(* Logix 5000 project; controller SX_V040001_C001 vendor 1 type 14 code 77 rev 16.22; software revision 16.04; part 32 of 35 *)
(* tags used below, declared in another part *)
   ALL_KINDS : INT[90];
   PARAMETER : INT[501];
   pointer_recipe_test : DINT;
(* MainProgram, continued *)

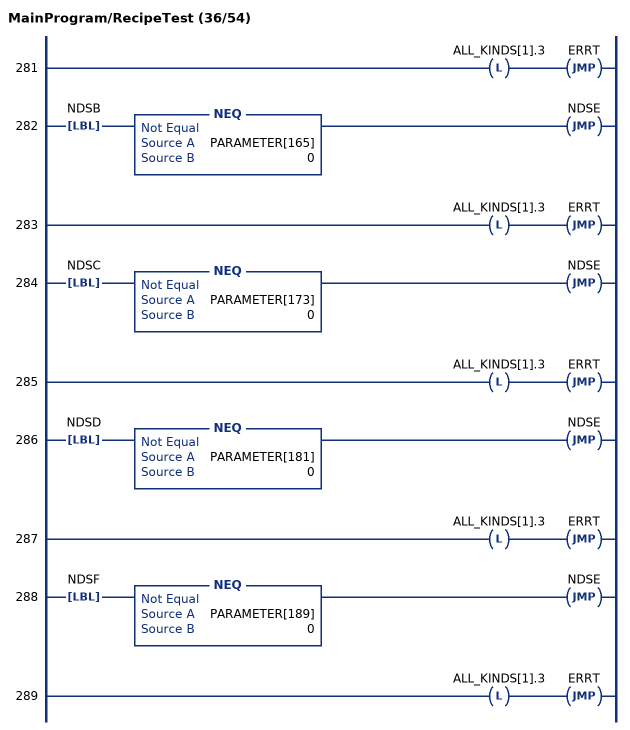
   [picture p701: MainProgram/RecipeTest rungs 281-289]
   281: OTL(ALL_KINDS[1].3)JMP(ERRT);
   282: LBL(NDSB)NEQ(PARAMETER[165],0)JMP(NDSE);
   283: OTL(ALL_KINDS[1].3)JMP(ERRT);
   284: LBL(NDSC)NEQ(PARAMETER[173],0)JMP(NDSE);
   285: OTL(ALL_KINDS[1].3)JMP(ERRT);
   286: LBL(NDSD)NEQ(PARAMETER[181],0)JMP(NDSE);
   287: OTL(ALL_KINDS[1].3)JMP(ERRT);
   288: LBL(NDSF)NEQ(PARAMETER[189],0)JMP(NDSE);
   289: OTL(ALL_KINDS[1].3)JMP(ERRT);
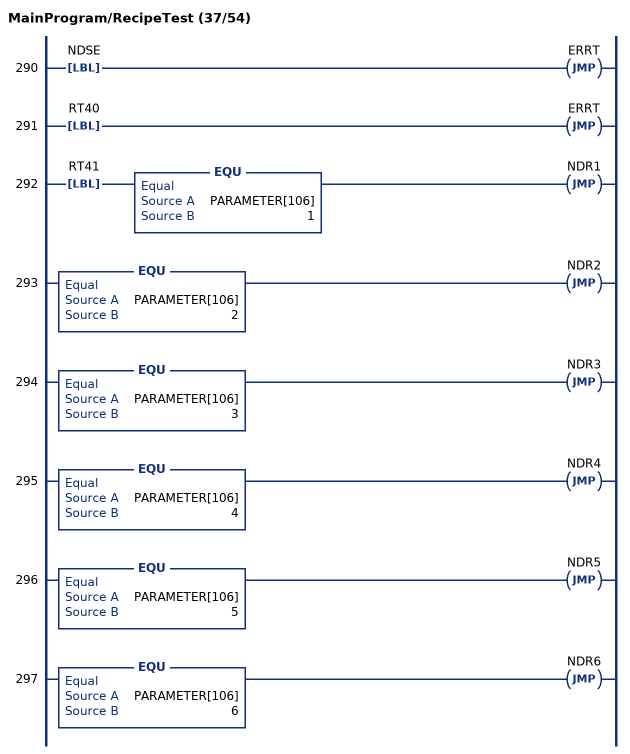
   290: LBL(NDSE)JMP(ERRT);
   291: LBL(RT40)JMP(ERRT);
   292: LBL(RT41)EQU(PARAMETER[106],1)JMP(NDR1);
   293: EQU(PARAMETER[106],2)JMP(NDR2);
   294: EQU(PARAMETER[106],3)JMP(NDR3);
   295: EQU(PARAMETER[106],4)JMP(NDR4);
   296: EQU(PARAMETER[106],5)JMP(NDR5);
   297: EQU(PARAMETER[106],6)JMP(NDR6);
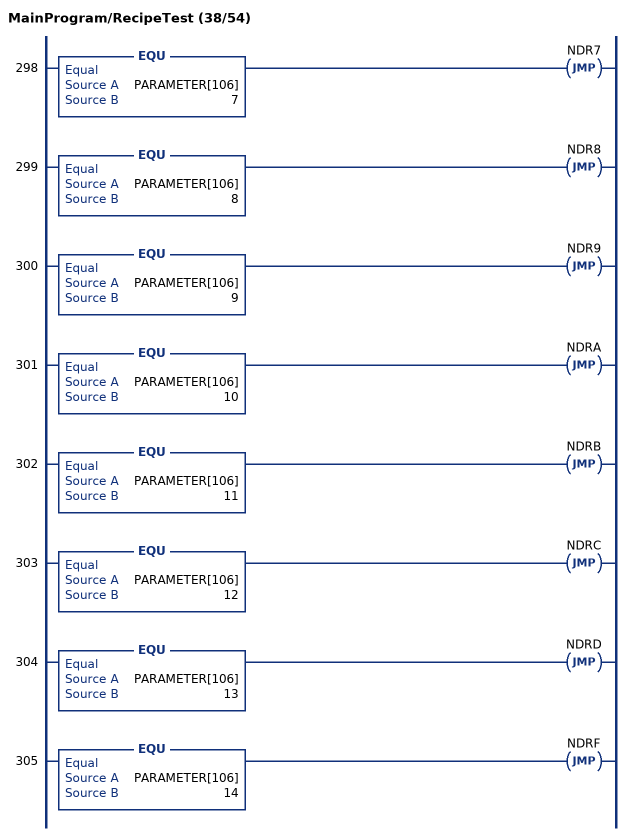
   298: EQU(PARAMETER[106],7)JMP(NDR7);
   299: EQU(PARAMETER[106],8)JMP(NDR8);
   300: EQU(PARAMETER[106],9)JMP(NDR9);
   301: EQU(PARAMETER[106],10)JMP(NDRA);
   302: EQU(PARAMETER[106],11)JMP(NDRB);
   303: EQU(PARAMETER[106],12)JMP(NDRC);
   304: EQU(PARAMETER[106],13)JMP(NDRD);
   305: EQU(PARAMETER[106],14)JMP(NDRF);
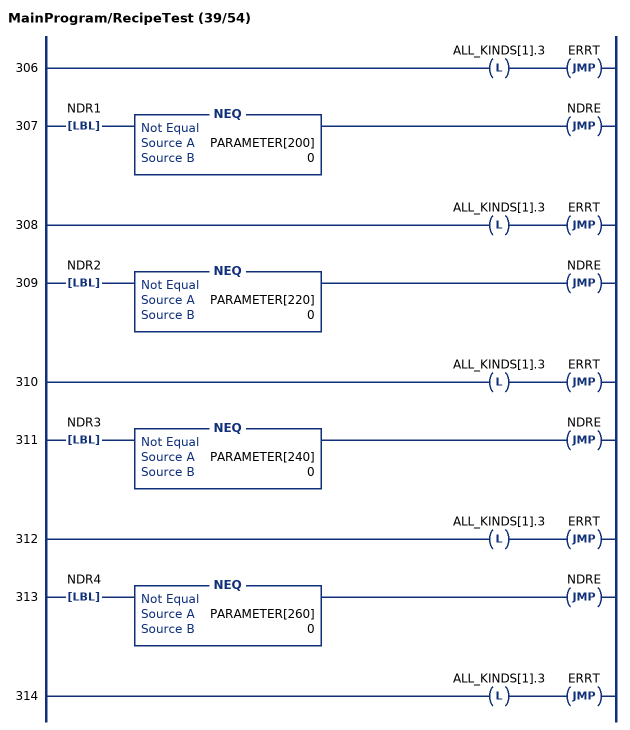
   306: OTL(ALL_KINDS[1].3)JMP(ERRT);
   307: LBL(NDR1)NEQ(PARAMETER[200],0)JMP(NDRE);
   308: OTL(ALL_KINDS[1].3)JMP(ERRT);
   309: LBL(NDR2)NEQ(PARAMETER[220],0)JMP(NDRE);
   310: OTL(ALL_KINDS[1].3)JMP(ERRT);
   311: LBL(NDR3)NEQ(PARAMETER[240],0)JMP(NDRE);
   312: OTL(ALL_KINDS[1].3)JMP(ERRT);
   313: LBL(NDR4)NEQ(PARAMETER[260],0)JMP(NDRE);
   314: OTL(ALL_KINDS[1].3)JMP(ERRT);
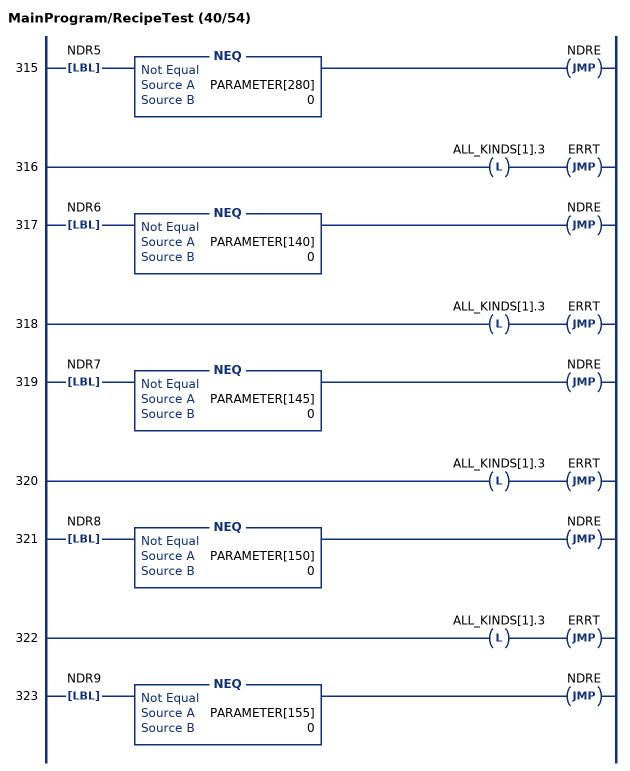
   315: LBL(NDR5)NEQ(PARAMETER[280],0)JMP(NDRE);
   316: OTL(ALL_KINDS[1].3)JMP(ERRT);
   317: LBL(NDR6)NEQ(PARAMETER[140],0)JMP(NDRE);
   318: OTL(ALL_KINDS[1].3)JMP(ERRT);
   319: LBL(NDR7)NEQ(PARAMETER[145],0)JMP(NDRE);
   320: OTL(ALL_KINDS[1].3)JMP(ERRT);
   321: LBL(NDR8)NEQ(PARAMETER[150],0)JMP(NDRE);
   322: OTL(ALL_KINDS[1].3)JMP(ERRT);
   323: LBL(NDR9)NEQ(PARAMETER[155],0)JMP(NDRE);
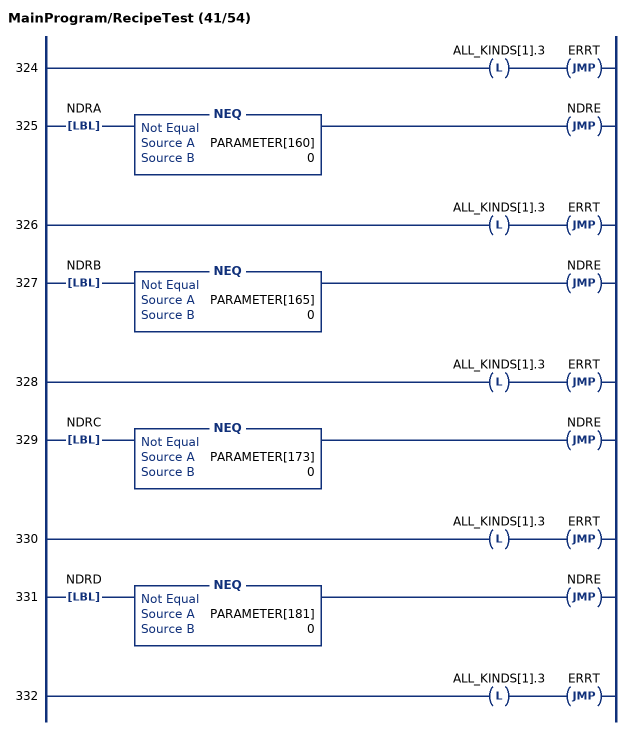
   324: OTL(ALL_KINDS[1].3)JMP(ERRT);
   325: LBL(NDRA)NEQ(PARAMETER[160],0)JMP(NDRE);
   326: OTL(ALL_KINDS[1].3)JMP(ERRT);
   327: LBL(NDRB)NEQ(PARAMETER[165],0)JMP(NDRE);
   328: OTL(ALL_KINDS[1].3)JMP(ERRT);
   329: LBL(NDRC)NEQ(PARAMETER[173],0)JMP(NDRE);
   330: OTL(ALL_KINDS[1].3)JMP(ERRT);
   331: LBL(NDRD)NEQ(PARAMETER[181],0)JMP(NDRE);
   332: OTL(ALL_KINDS[1].3)JMP(ERRT);
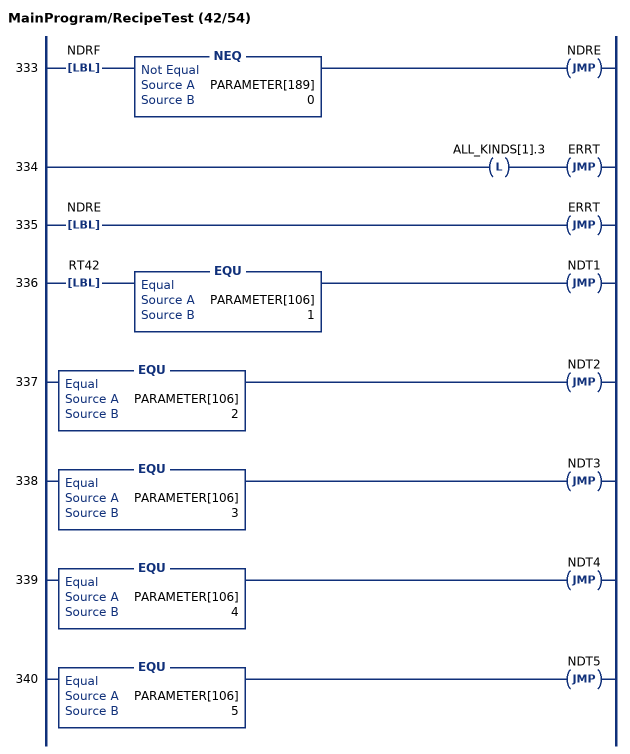
   333: LBL(NDRF)NEQ(PARAMETER[189],0)JMP(NDRE);
   334: OTL(ALL_KINDS[1].3)JMP(ERRT);
   335: LBL(NDRE)JMP(ERRT);
   336: LBL(RT42)EQU(PARAMETER[106],1)JMP(NDT1);
   337: EQU(PARAMETER[106],2)JMP(NDT2);
   338: EQU(PARAMETER[106],3)JMP(NDT3);
   339: EQU(PARAMETER[106],4)JMP(NDT4);
   340: EQU(PARAMETER[106],5)JMP(NDT5);
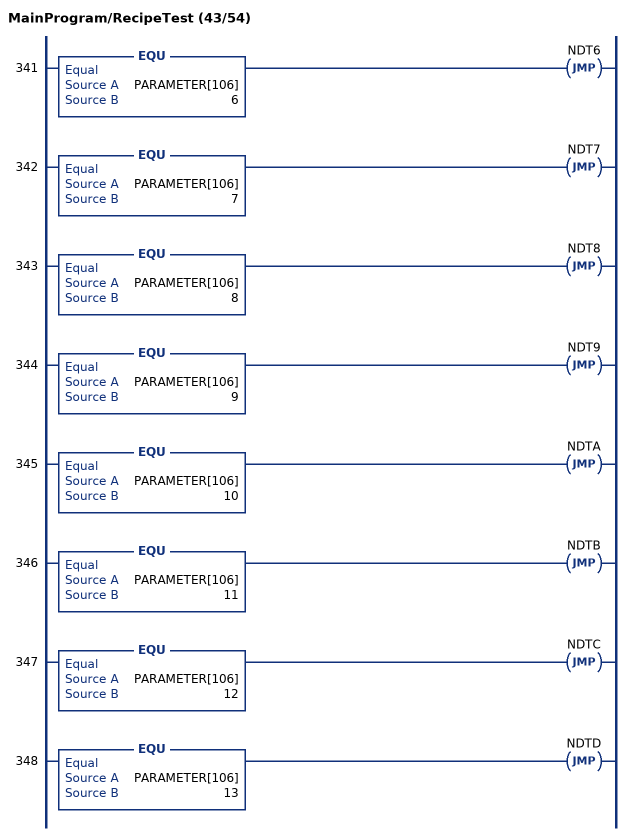
   341: EQU(PARAMETER[106],6)JMP(NDT6);
   342: EQU(PARAMETER[106],7)JMP(NDT7);
   343: EQU(PARAMETER[106],8)JMP(NDT8);
   344: EQU(PARAMETER[106],9)JMP(NDT9);
   345: EQU(PARAMETER[106],10)JMP(NDTA);
   346: EQU(PARAMETER[106],11)JMP(NDTB);
   347: EQU(PARAMETER[106],12)JMP(NDTC);
   348: EQU(PARAMETER[106],13)JMP(NDTD);
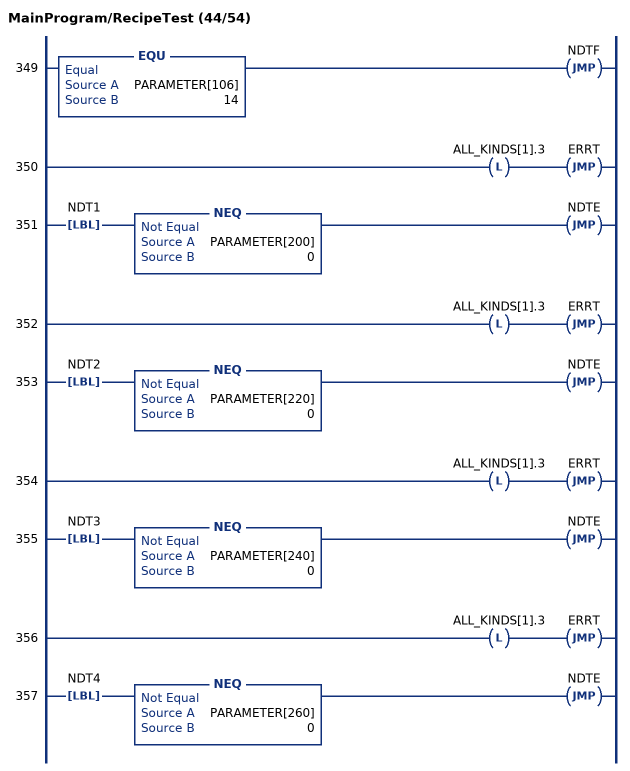
   349: EQU(PARAMETER[106],14)JMP(NDTF);
   350: OTL(ALL_KINDS[1].3)JMP(ERRT);
   351: LBL(NDT1)NEQ(PARAMETER[200],0)JMP(NDTE);
   352: OTL(ALL_KINDS[1].3)JMP(ERRT);
   353: LBL(NDT2)NEQ(PARAMETER[220],0)JMP(NDTE);
   354: OTL(ALL_KINDS[1].3)JMP(ERRT);
   355: LBL(NDT3)NEQ(PARAMETER[240],0)JMP(NDTE);
   356: OTL(ALL_KINDS[1].3)JMP(ERRT);
   357: LBL(NDT4)NEQ(PARAMETER[260],0)JMP(NDTE);
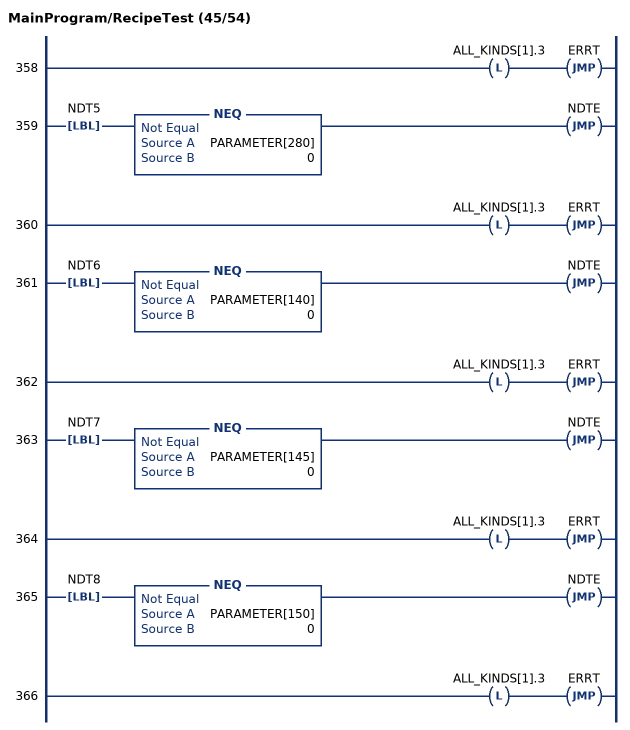
   358: OTL(ALL_KINDS[1].3)JMP(ERRT);
   359: LBL(NDT5)NEQ(PARAMETER[280],0)JMP(NDTE);
   360: OTL(ALL_KINDS[1].3)JMP(ERRT);
   361: LBL(NDT6)NEQ(PARAMETER[140],0)JMP(NDTE);
   362: OTL(ALL_KINDS[1].3)JMP(ERRT);
   363: LBL(NDT7)NEQ(PARAMETER[145],0)JMP(NDTE);
   364: OTL(ALL_KINDS[1].3)JMP(ERRT);
   365: LBL(NDT8)NEQ(PARAMETER[150],0)JMP(NDTE);
   366: OTL(ALL_KINDS[1].3)JMP(ERRT);
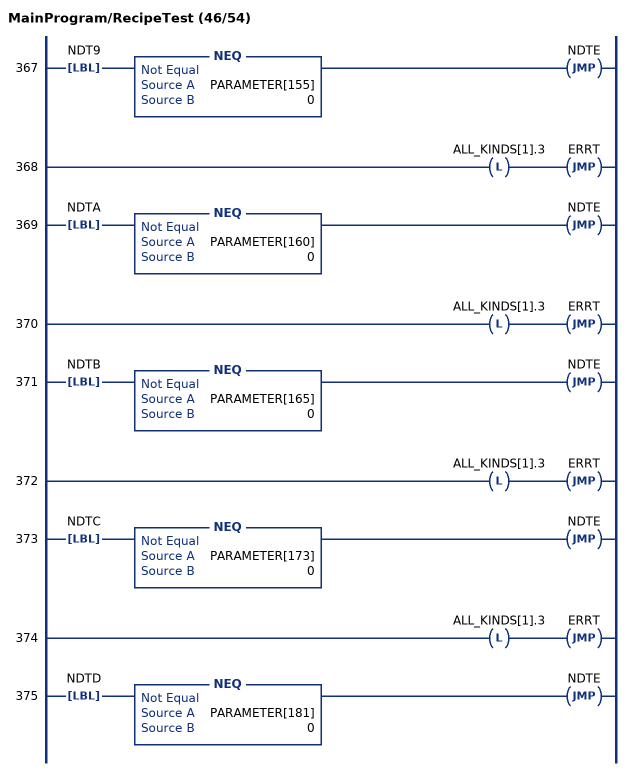
   367: LBL(NDT9)NEQ(PARAMETER[155],0)JMP(NDTE);
   368: OTL(ALL_KINDS[1].3)JMP(ERRT);
   369: LBL(NDTA)NEQ(PARAMETER[160],0)JMP(NDTE);
   370: OTL(ALL_KINDS[1].3)JMP(ERRT);
   371: LBL(NDTB)NEQ(PARAMETER[165],0)JMP(NDTE);
   372: OTL(ALL_KINDS[1].3)JMP(ERRT);
   373: LBL(NDTC)NEQ(PARAMETER[173],0)JMP(NDTE);
   374: OTL(ALL_KINDS[1].3)JMP(ERRT);
   375: LBL(NDTD)NEQ(PARAMETER[181],0)JMP(NDTE);
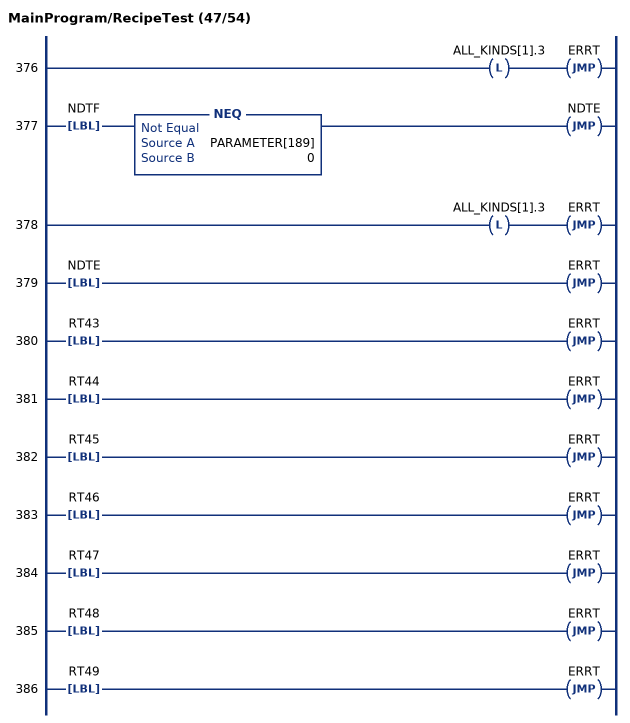
   376: OTL(ALL_KINDS[1].3)JMP(ERRT);
   377: LBL(NDTF)NEQ(PARAMETER[189],0)JMP(NDTE);
   378: OTL(ALL_KINDS[1].3)JMP(ERRT);
   379: LBL(NDTE)JMP(ERRT);
   380: LBL(RT43)JMP(ERRT);
   381: LBL(RT44)JMP(ERRT);
   382: LBL(RT45)JMP(ERRT);
   383: LBL(RT46)JMP(ERRT);
   384: LBL(RT47)JMP(ERRT);
   385: LBL(RT48)JMP(ERRT);
   386: LBL(RT49)JMP(ERRT);
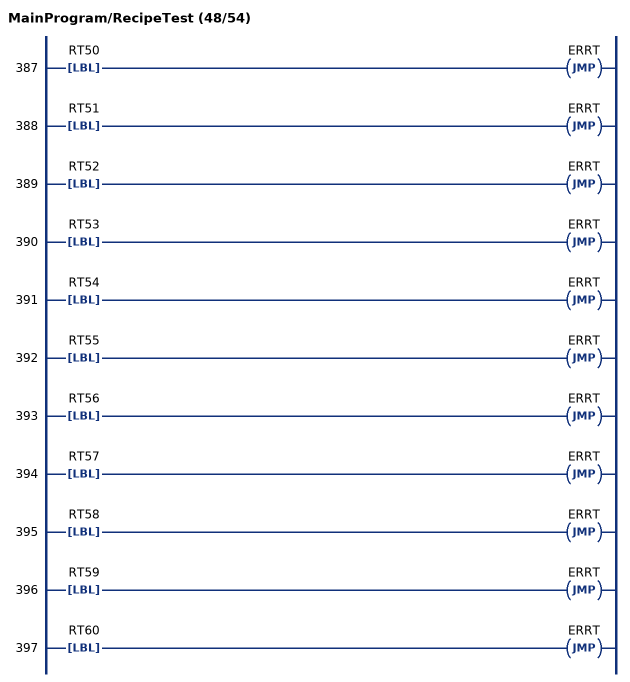
   387: LBL(RT50)JMP(ERRT);
   388: LBL(RT51)JMP(ERRT);
   389: LBL(RT52)JMP(ERRT);
   390: LBL(RT53)JMP(ERRT);
   391: LBL(RT54)JMP(ERRT);
   392: LBL(RT55)JMP(ERRT);
   393: LBL(RT56)JMP(ERRT);
   394: LBL(RT57)JMP(ERRT);
   395: LBL(RT58)JMP(ERRT);
   396: LBL(RT59)JMP(ERRT);
   397: LBL(RT60)JMP(ERRT);
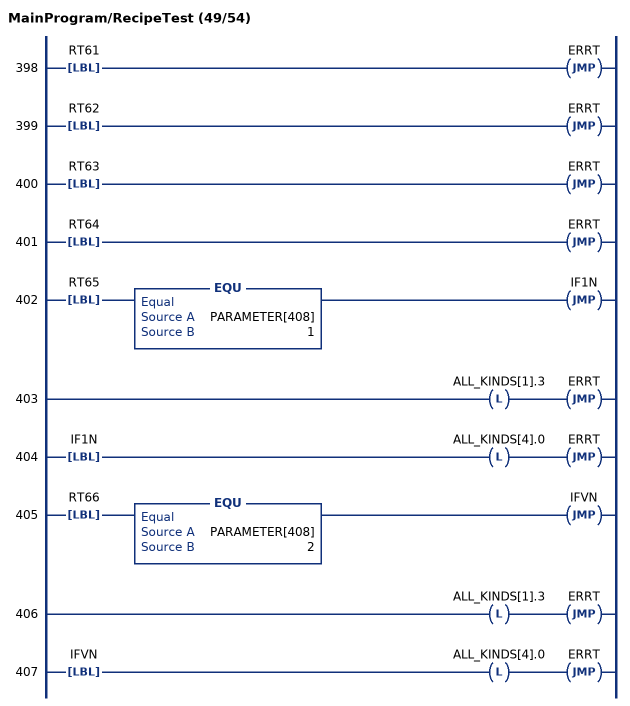
   398: LBL(RT61)JMP(ERRT);
   399: LBL(RT62)JMP(ERRT);
   400: LBL(RT63)JMP(ERRT);
   401: LBL(RT64)JMP(ERRT);
   402: LBL(RT65)EQU(PARAMETER[408],1)JMP(IF1N);
   403: OTL(ALL_KINDS[1].3)JMP(ERRT);
   404: LBL(IF1N)OTL(ALL_KINDS[4].0)JMP(ERRT);
   405: LBL(RT66)EQU(PARAMETER[408],2)JMP(IFVN);
   406: OTL(ALL_KINDS[1].3)JMP(ERRT);
   407: LBL(IFVN)OTL(ALL_KINDS[4].0)JMP(ERRT);
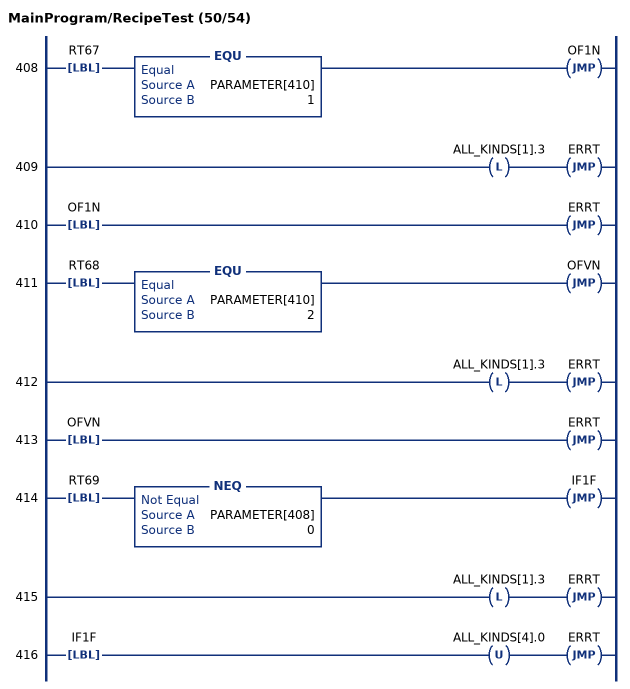
   408: LBL(RT67)EQU(PARAMETER[410],1)JMP(OF1N);
   409: OTL(ALL_KINDS[1].3)JMP(ERRT);
   410: LBL(OF1N)JMP(ERRT);
   411: LBL(RT68)EQU(PARAMETER[410],2)JMP(OFVN);
   412: OTL(ALL_KINDS[1].3)JMP(ERRT);
   413: LBL(OFVN)JMP(ERRT);
   414: LBL(RT69)NEQ(PARAMETER[408],0)JMP(IF1F);
   415: OTL(ALL_KINDS[1].3)JMP(ERRT);
   416: LBL(IF1F)OTU(ALL_KINDS[4].0)JMP(ERRT);
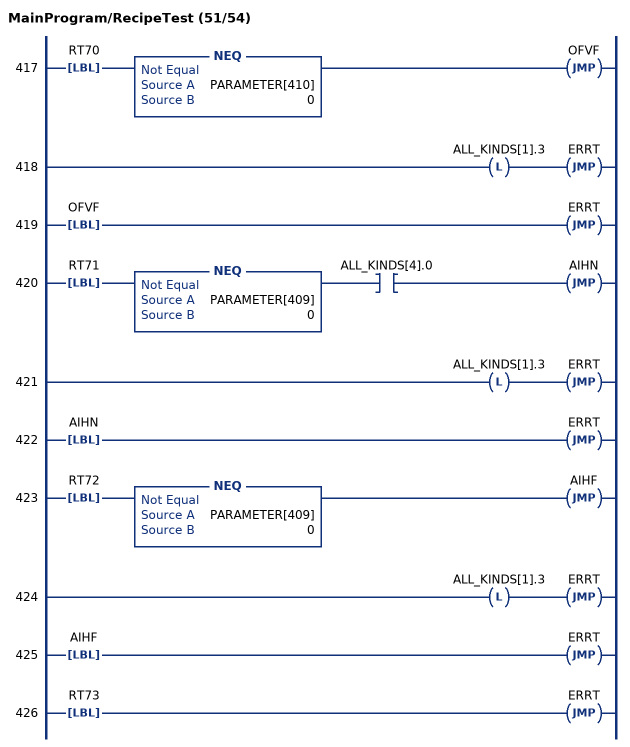
   417: LBL(RT70)NEQ(PARAMETER[410],0)JMP(OFVF);
   418: OTL(ALL_KINDS[1].3)JMP(ERRT);
   419: LBL(OFVF)JMP(ERRT);
   420: LBL(RT71)NEQ(PARAMETER[409],0)XIC(ALL_KINDS[4].0)JMP(AIHN);
   421: OTL(ALL_KINDS[1].3)JMP(ERRT);
   422: LBL(AIHN)JMP(ERRT);
   423: LBL(RT72)NEQ(PARAMETER[409],0)JMP(AIHF);
   424: OTL(ALL_KINDS[1].3)JMP(ERRT);
   425: LBL(AIHF)JMP(ERRT);
   426: LBL(RT73)JMP(ERRT);
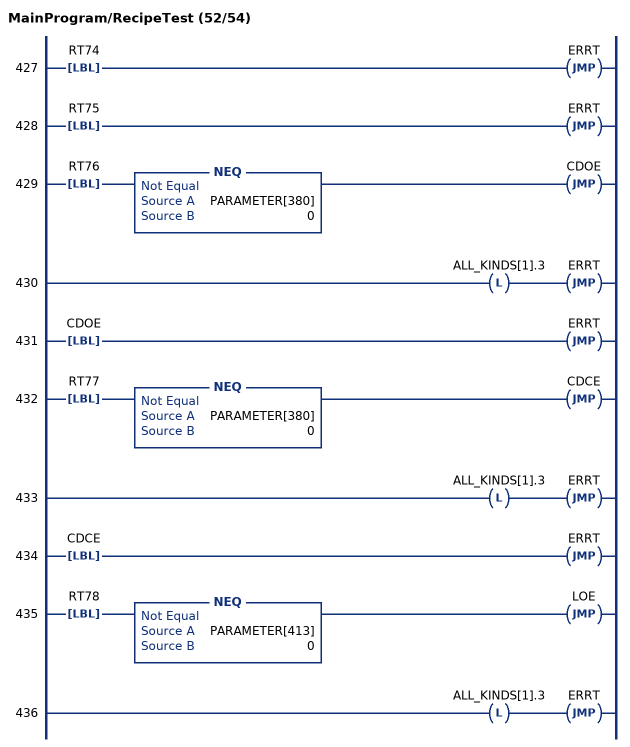
   427: LBL(RT74)JMP(ERRT);
   428: LBL(RT75)JMP(ERRT);
   429: LBL(RT76)NEQ(PARAMETER[380],0)JMP(CDOE);
   430: OTL(ALL_KINDS[1].3)JMP(ERRT);
   431: LBL(CDOE)JMP(ERRT);
   432: LBL(RT77)NEQ(PARAMETER[380],0)JMP(CDCE);
   433: OTL(ALL_KINDS[1].3)JMP(ERRT);
   434: LBL(CDCE)JMP(ERRT);
   435: LBL(RT78)NEQ(PARAMETER[413],0)JMP(LOE);
   436: OTL(ALL_KINDS[1].3)JMP(ERRT);
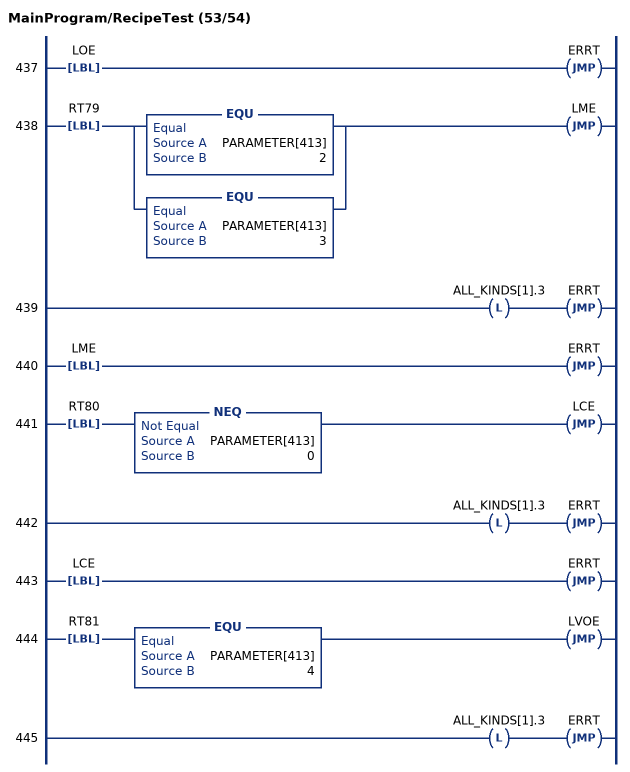
   437: LBL(LOE)JMP(ERRT);
   438: LBL(RT79)[EQU(PARAMETER[413],2) ,EQU(PARAMETER[413],3) ]JMP(LME);
   439: OTL(ALL_KINDS[1].3)JMP(ERRT);
   440: LBL(LME)JMP(ERRT);
   441: LBL(RT80)NEQ(PARAMETER[413],0)JMP(LCE);
   442: OTL(ALL_KINDS[1].3)JMP(ERRT);
   443: LBL(LCE)JMP(ERRT);
   444: LBL(RT81)EQU(PARAMETER[413],4)JMP(LVOE);
   445: OTL(ALL_KINDS[1].3)JMP(ERRT);
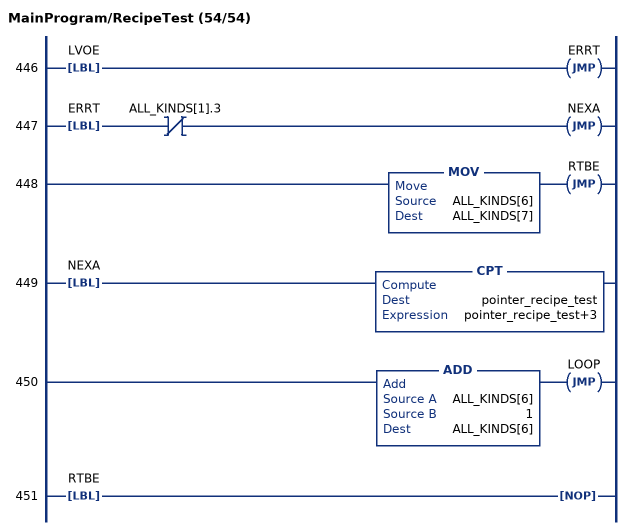
   446: LBL(LVOE)JMP(ERRT);
   447: LBL(ERRT)XIO(ALL_KINDS[1].3)JMP(NEXA);
   448: MOV(ALL_KINDS[6],ALL_KINDS[7])JMP(RTBE);
   449: LBL(NEXA)CPT(pointer_recipe_test,pointer_recipe_test+3);
   450: ADD(ALL_KINDS[6],1,ALL_KINDS[6])JMP(LOOP);
   451: LBL(RTBE)NOP();
END_ROUTINE
